FUNCTION_BLOCK ConvertAnyToString_TEST EXTENDS TcUnit.FB_TestSuite

ConvertAnyByteToString();
ConvertAnyDateAndTimeToString();
ConvertAnyDateToString();
ConvertAnyDINTToString();
ConvertAnyDTToString();
ConvertAnyINTToString();
ConvertAnyLINTToString();
//ConvertAnyLRealToString();
ConvertAnyLWordToString();
ConvertAnyRealToString();
ConvertAnySINTToString();
ConvertAnyStringToString();
ConvertAnyTimeToString();
ConvertAnyTODToString();
ConvertAnyUDINTToString();
ConvertAnyUINTToString();
ConvertAnyULINTToString();
ConvertAnyUSINTToString();
ConvertAnyWordToString();
ConvertAnyWStringToString();

METHOD ConvertAnyByteToString : BOOL
VAR
  inputs : ARRAY[1..4] OF BYTE := [0, 1, 128, 255];
  expectedValues : ARRAY[1..4] OF STRING := ['0', '1', '128', '255'];
  results : ARRAY[1..4] OF STRING;
  i: INT;
END_VAR
TEST('ConvertAnyByteToString');
 
FOR i := 1 TO 4 DO
  results[i] := AnyToString(inputs[i]);
  AssertEquals(Expected := expectedValues[i],
             Actual := results[i],
             Message := FormatResult(expectedValues[i], results[i])); 
END_FOR
 
TEST_FINISHED();
END_METHOD

METHOD ConvertAnyDateAndTimeToString : BOOL
VAR
  input : DATE_AND_TIME := DT#1970-01-01-00:00;
  result : STRING;
  expected : STRING := 'DT#1970-01-01-00:00:00';
END_VAR
TEST('ConvertAnyDateAndTimeToString');
 
result := AnyToString(input);
 
AssertEquals(Expected := expected,
             Actual := result,
             Message := FormatResult(expected, result));
 
TEST_FINISHED();
END_METHOD

METHOD ConvertAnyDateToString : BOOL
VAR
  input : DATE := D#1970-01-01;
  result : STRING;
  expected : STRING := 'D#1970-01-01';
END_VAR
TEST('ConvertAnyDateToString');
 
result := AnyToString(input);
 
AssertEquals(Expected := expected,
             Actual := result,
             Message := FormatResult(expected, result));
 
TEST_FINISHED();
END_METHOD

METHOD ConvertAnyDINTToString : BOOL
VAR
  inputs : ARRAY[1..7] OF DINT := [-2147483648, -1073741824, -1, 0, 1, 1073741824, 2147483647];
  expectedValues : ARRAY[1..7] OF STRING := ['-2147483648', '-1073741824', '-1', '0', '1', '1073741824', '2147483647'];
  results : ARRAY[1..7] OF STRING;
  i: INT;
END_VAR
TEST('ConvertAnyDINTToString');
 
FOR i := 1 TO 7 DO
  results[i] := AnyToString(inputs[i]);
  AssertEquals(Expected := expectedValues[i],
             Actual := results[i],
             Message := FormatResult(expectedValues[i], results[i])); 
END_FOR

TEST_FINISHED();
END_METHOD

METHOD ConvertAnyDTToString : BOOL
VAR
  input : DT := DT#1970-01-01-00:00;
  result : STRING;
  expected : STRING := 'DT#1970-01-01-00:00:00';
END_VAR
TEST('ConvertAnyDTToString');
 
result := AnyToString(input);
 
AssertEquals(Expected := expected,
             Actual := result,
             Message := FormatResult(expected, result));
 
TEST_FINISHED();
END_METHOD

METHOD ConvertAnyDWordToString : BOOL
VAR
  inputs : ARRAY[1..4] OF DWORD := [0, 1, 2147483647, 4294967295];
  expectedValues : ARRAY[1..4] OF STRING := ['0', '1', '2147483647', '4294967295'];
  results : ARRAY[1..4] OF STRING;
  i: INT;
END_VAR
TEST('ConvertAnyDWordToString');
 
FOR i := 1 TO 4 DO
  results[i] := AnyToString(inputs[i]);
  AssertEquals(Expected := expectedValues[i],
             Actual := results[i],
             Message := FormatResult(expectedValues[i], results[i])); 
END_FOR
 
TEST_FINISHED();
END_METHOD

METHOD ConvertAnyINTToString : BOOL
VAR
  inputs : ARRAY[1..7] OF INT := [-32768, -18000, -1, 0, 1, 18000, 32767];
  expectedValues : ARRAY[1..7] OF STRING := ['-32768', '-18000', '-1', '0', '1', '18000', '32767'];
  results : ARRAY[1..7] OF STRING;
  i: INT;
END_VAR
TEST('ConvertAnyINTToString');

FOR i := 1 TO 7 DO
  results[i] := AnyToString(inputs[i]);
  AssertEquals(Expected := expectedValues[i],
             Actual := results[i],
             Message := FormatResult(expectedValues[i], results[i])); 
END_FOR
      
TEST_FINISHED();
END_METHOD

METHOD ConvertAnyLINTToString : BOOL
VAR
  inputs : ARRAY[1..7] OF LINT := [-2147483648, -18000, -1, 0, 1, 18000, 2147483648];
  expectedValues : ARRAY[1..7] OF STRING := ['-2147483648', '-18000', '-1', '0', '1', '18000', '2147483648'];
  results : ARRAY[1..7] OF STRING;
  i: INT;
END_VAR
TEST('ConvertAnyLINTToString');
 
FOR i := 1 TO 7 DO
  results[i] := AnyToString(inputs[i]);
  AssertEquals(Expected := expectedValues[i],
             Actual := results[i],
             Message := FormatResult(expectedValues[i], results[i])); 
END_FOR
 
TEST_FINISHED();
END_METHOD

METHOD ConvertAnyLRealToString : BOOL
VAR
  inputs : ARRAY[1..5] OF LREAL := [-1.7976931348623157E+308, -4.94065645841247E-324, 0, 4.94065645841247E-324, 1.7976931348623157E+308];
  expectedValues : ARRAY[1..5] OF STRING := ['-1.7976931348623157E308', '-4.94065645841247E324', '0.0', '4.94065645841247E324', '1.7976931348623157E308'];
  results : ARRAY[1..5] OF STRING;
  i: INT;
END_VAR
TEST('ConvertAnyRealToString');
 
FOR i := 1 TO 5 DO
  results[i] := AnyToString(inputs[i]);
  AssertEquals(Expected := expectedValues[i],
             Actual := results[i],
             Message := FormatResult(expectedValues[i], results[i])); 
END_FOR
 
TEST_FINISHED();
END_METHOD

METHOD ConvertAnyLWordToString : BOOL
VAR
  inputs : ARRAY[1..4] OF LWORD := [0, 1, 2147483647, 4294967295];
  expectedValues : ARRAY[1..4] OF STRING := ['0', '1', '2147483647', '4294967295'];
  results : ARRAY[1..4] OF STRING;
  i: INT;
END_VAR
TEST('ConvertAnyLWordToString');
 
FOR i := 1 TO 4 DO
  results[i] := AnyToString(inputs[i]);
  AssertEquals(Expected := expectedValues[i],
             Actual := results[i],
             Message := FormatResult(expectedValues[i], results[i])); 
END_FOR

TEST_FINISHED();
END_METHOD

METHOD ConvertAnyRealToString : BOOL
VAR
  inputs : ARRAY[1..5] OF REAL := [-3.402823E+38, -1.0, 0, 1.0, 3.402823E+38];
  expectedValues : ARRAY[1..5] OF STRING := ['-3.402823E38', '-1.0', '0.0', '1.0', '3.402823E38'];
  results : ARRAY[1..5] OF STRING;
  i: INT;
END_VAR
TEST('ConvertAnyRealToString');
 
FOR i := 1 TO 5 DO
  results[i] := AnyToString(inputs[i]);
  AssertEquals(Expected := expectedValues[i],
             Actual := results[i],
             Message := FormatResult(expectedValues[i], results[i])); 
END_FOR
 
TEST_FINISHED();
END_METHOD

METHOD ConvertAnySINTToString : BOOL
VAR
  inputs : ARRAY[1..5] OF SINT := [-128, -1, 0, 1, 127];
  expectedValues : ARRAY[1..5] OF STRING := ['-128', '-1', '0', '1', '127'];
  results : ARRAY[1..5] OF STRING;
  i: INT;
END_VAR
TEST('ConvertAnySINTToString');
 
FOR i := 1 TO 5 DO
  results[i] := AnyToString(inputs[i]);
  AssertEquals(Expected := expectedValues[i],
             Actual := results[i],
             Message := FormatResult(expectedValues[i], results[i])); 
END_FOR
 
TEST_FINISHED();
END_METHOD

METHOD ConvertAnyStringToString : BOOL
VAR
  input : STRING := 'Hallo';
  result : STRING;
  expected : STRING := 'Hallo';
END_VAR
TEST('ConvertAnyStringToString');
 
result := AnyToString(input);
 
AssertEquals(Expected := expected,
             Actual := result,
             Message := FormatResult(expected, result));
 
TEST_FINISHED();
END_METHOD

METHOD ConvertAnyTimeToString : BOOL
VAR
  input : TIME := T#49D17H2M47S295MS;
  result : STRING;
  expected : STRING := 'T#49d17h2m47s295ms';
END_VAR
TEST('ConvertAnyTimeToString');
 
result := AnyToString(input);
 
AssertEquals(Expected := expected,
             Actual := result,
             Message := FormatResult(expected, result));
 
TEST_FINISHED();
END_METHOD

METHOD ConvertAnyTODToString : BOOL
VAR
  input : TOD := TOD#11:02:47.295;
  result : STRING;
  expected : STRING := 'TOD#11:02:47.295';
END_VAR
TEST('ConvertAnyTODToString');
 
result := AnyToString(input);
 
AssertEquals(Expected := expected,
             Actual := result,
             Message := FormatResult(expected, result));
 
TEST_FINISHED();
END_METHOD

METHOD ConvertAnyUDINTToString : BOOL
VAR
  inputs : ARRAY[1..3] OF UDINT := [0, 1, 4294967295];
  expectedValues : ARRAY[1..3] OF STRING := ['0', '1', '4294967295'];
  results : ARRAY[1..3] OF STRING;
  i: INT;
END_VAR
TEST('ConvertAnyUDINTToString');

FOR i := 1 TO 3 DO
  results[i] := AnyToString(inputs[i]);
  AssertEquals(Expected := expectedValues[i],
             Actual := results[i],
             Message := FormatResult(expectedValues[i], results[i])); 
END_FOR
 
TEST_FINISHED();
END_METHOD

METHOD ConvertAnyUINTToString : BOOL
VAR
  inputs : ARRAY[1..3] OF UINT := [0, 1, 65535];
  expectedValues : ARRAY[1..3] OF STRING := ['0', '1', '65535'];
  results : ARRAY[1..3] OF STRING;
  i: INT;
END_VAR
TEST('ConvertAnyUINTToString');
 
FOR i := 1 TO 3 DO
  results[i] := AnyToString(inputs[i]);
  AssertEquals(Expected := expectedValues[i],
             Actual := results[i],
             Message := FormatResult(expectedValues[i], results[i])); 
END_FOR
 
TEST_FINISHED();
END_METHOD

METHOD ConvertAnyULINTToString : BOOL
VAR
  inputs : ARRAY[1..3] OF ULINT := [0, 1, 4294967295];
  expectedValues : ARRAY[1..3] OF STRING := ['0', '1', '4294967295'];
  results : ARRAY[1..3] OF STRING;
  i: INT;
END_VAR
TEST('ConvertAnyULINTToString');
 
FOR i := 1 TO 3 DO
  results[i] := AnyToString(inputs[i]);
  AssertEquals(Expected := expectedValues[i],
             Actual := results[i],
             Message := FormatResult(expectedValues[i], results[i])); 
END_FOR
 
TEST_FINISHED();
END_METHOD

METHOD ConvertAnyUSINTToString : BOOL
VAR
  inputs : ARRAY[1..3] OF USINT := [0, 1, 255];
  expectedValues : ARRAY[1..3] OF STRING := ['0', '1', '255'];
  results : ARRAY[1..3] OF STRING;
  i: INT;
END_VAR
TEST('ConvertAnyUSINTToString');
 
FOR i := 1 TO 3 DO
  results[i] := AnyToString(inputs[i]);
  AssertEquals(Expected := expectedValues[i],
             Actual := results[i],
             Message := FormatResult(expectedValues[i], results[i])); 
END_FOR
 
TEST_FINISHED();
END_METHOD

METHOD ConvertAnyWordToString : BOOL
VAR
  inputs : ARRAY[1..3] OF WORD := [0, 1, 65535];
  expectedValues : ARRAY[1..3] OF STRING := ['0', '1', '65535'];
  results : ARRAY[1..3] OF STRING;
  i: INT;
END_VAR
TEST('ConvertAnyWordToString');
 
FOR i := 1 TO 3 DO
  results[i] := AnyToString(inputs[i]);
  AssertEquals(Expected := expectedValues[i],
             Actual := results[i],
             Message := FormatResult(expectedValues[i], results[i])); 
END_FOR
 
TEST_FINISHED();
END_METHOD

METHOD ConvertAnyWStringToString : BOOL
VAR
  input : WSTRING := "Hallo";
  result : STRING;
  expected : STRING := 'Hallo';
END_VAR
TEST('ConvertAnyWStringToString');
 
result := AnyToString(input);
 
AssertEquals(Expected := expected,
             Actual := result,
             Message := FormatResult(expected, result));
 
TEST_FINISHED();
END_METHOD

METHOD PRIVATE FormatResult : STRING
VAR_INPUT
  Expected : STRING;
  Result : STRING;
END_VAR
FormatResult := Tc2_Standard.CONCAT('Conversion failed. Expected: ', Tc2_Standard.CONCAT(Expected, Tc2_Standard.CONCAT(' - Result: ', Result)));
END_METHOD

END_FUNCTION_BLOCK

(* stored: Version 1.1.0.1
   POU ConvertAnyToString_TEST: Id {8723bf95-47c2-4342-9746-8c558da116aa}, SpecialFunc None
   Method ConvertAnyByteToString: Id {6a4de533-1ff4-4300-bd1b-aa9dee141478}
   Method ConvertAnyDateAndTimeToString: Id {9ec8d9a4-8741-4865-a722-ba411337f891}
   Method ConvertAnyDateToString: Id {01dc3069-8329-4d56-baac-d69a1aaef399}
   Method ConvertAnyDINTToString: Id {9bf59e16-f1e6-45ac-a807-e1d1de1d7a2c}
   Method ConvertAnyDTToString: Id {6f1e9768-4e40-4c59-bb14-df57394138b5}
   Method ConvertAnyDWordToString: Id {4f8362c2-1bc1-4575-a937-4e7d8af79721}
   Method ConvertAnyINTToString: Id {03af596d-48bd-41ed-bda7-49b17c1fbeb2}
   Method ConvertAnyLINTToString: Id {8e7df9bc-31be-419d-beb5-aa1f224ebdc7}
   Method ConvertAnyLRealToString: Id {42351668-e462-4446-aac6-670516acb622}
   Method ConvertAnyLWordToString: Id {db8455a2-4fe9-44ea-81da-61701a6999c0}
   Method ConvertAnyRealToString: Id {7dde6cfd-c6ff-45c1-80bc-3da59350d708}
   Method ConvertAnySINTToString: Id {0e12c253-d6dc-43ca-ad90-0a44d459c5a8}
   Method ConvertAnyStringToString: Id {878de958-8cc9-40c7-86f0-88d52c3b1291}
   Method ConvertAnyTimeToString: Id {a7ef71a7-444f-4dc1-955b-c0574355c4c6}
   Method ConvertAnyTODToString: Id {e06cf1c5-87e8-426a-9089-bc21534675bb}
   Method ConvertAnyUDINTToString: Id {3229ca76-3df9-44f7-aacd-19b8138d5651}
   Method ConvertAnyUINTToString: Id {ba193657-134b-49fe-8445-16bf4f0f5139}
   Method ConvertAnyULINTToString: Id {2eef74a8-d2ce-40e5-ada9-a977392f50d2}
   Method ConvertAnyUSINTToString: Id {54e44617-410b-411f-9440-d611d1294e71}
   Method ConvertAnyWordToString: Id {58d7c7a1-012a-4615-9b88-6f8dbc3301fc}
   Method ConvertAnyWStringToString: Id {4a04c330-3f68-4390-83b8-8e7e709d4d25}
   Method FormatResult: Id {dfc117b2-1e90-4366-99ce-6966d5be1d1d} *)
